//Error FB instance
EK1100_Error(
    En                  := TRUE,
    iTerminal_ID        := iTerminal_ID,
    bWcState            := FALSE,
    uiInfoData_State    := InfoData_State,
    pErrorSystem        := ErrorSystem,
    bError              => bError,
);

IF bError THEN
	sErrorMessage:=EK1100_Error.ErrorData.sErrorMessage;
ELSE
	sErrorMessage:='';
END_IF

END_FUNCTION_BLOCK

// ---- POUs/Data Type Conversion Functions/SCALE_REAL_TO_UDINT.TcPOU
FUNCTION SCALE_REAL_TO_UDINT : UDINT
VAR_INPUT
	I : REAL;
	Range_LL : REAL;
	Range_UL : REAL;
END_VAR
VAR
END_VAR

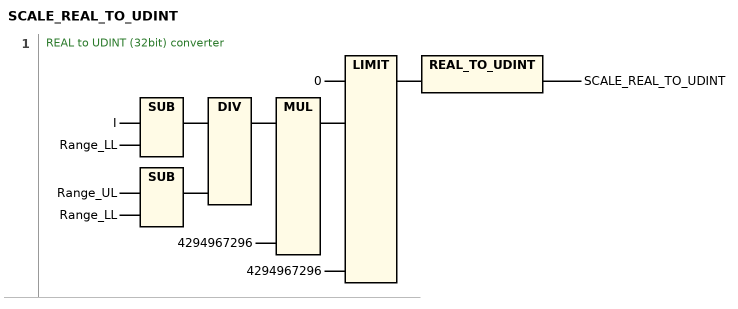
// NETWORK 1
// REAL to UDINT (32bit) converter
SCALE_REAL_TO_UDINT := REAL_TO_UDINT(LIMIT(0, ((I - Range_LL) / (Range_UL - Range_LL)) * 4294967296, 4294967296));

END_FUNCTION

// ---- POUs/Data Type Conversion Functions/SCALE_UDINT_TO_REAL.TcPOU
FUNCTION SCALE_UDINT_TO_REAL : REAL
VAR_INPUT
	I : UDINT;
	Range_LL : REAL;
	Range_UL : REAL;
END_VAR
VAR
END_VAR

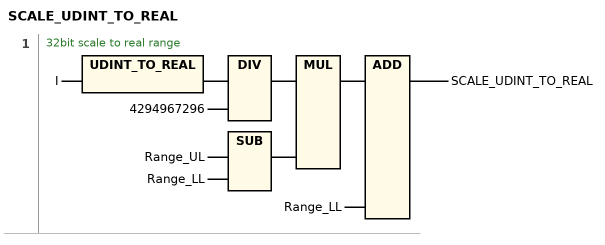
// NETWORK 1
// 32bit scale to real range
SCALE_UDINT_TO_REAL := (UDINT_TO_REAL(I) / 4294967296) * (Range_UL - Range_LL) + Range_LL;

END_FUNCTION

// ---- GlobalTextList.TcGTLO
TEXTLIST GlobalTextList
  561 = '   LocalMode'
  951 = '%2.2f'
  543 = '%2.4f'
  706 = '%i'
  940 = '%x'
  703 = 'Acknowledge'
  710 = 'Active:'
  952 = 'actPos'
  953 = 'actVel'
  110 = 'AXESMAX'
  107 = 'axisSel'
  945 = 'bBusy'
  950 = 'bBwEnabled'
  225 = 'bCommandAborted'
  946 = 'bDone'
  943 = 'bEnabled'
  941 = 'bError'
  102 = 'bExecute'
  949 = 'bFwEnabled'
  297 = 'bGeared'
  948 = 'bHomed'
  947 = 'bResetDone'
  944 = 'bWarning'
  704 = 'Clear All'
  986 = 'ehomeDirect'
  198 = 'eHomeToEncPulse_Bwd'
  510 = 'eHomeToEncPulse_Fwd'
  287 = 'eHomeToEncPulse_viaBwdLimit'
  683 = 'eHomeToEncPulse_viaFwdLimit'
  312 = 'eHomeToLimit_Bwd'
  635 = 'eHomeToLimit_Fwd'
  150 = 'eHomeToRef_Bwd'
  861 = 'eHomeToRef_Fwd'
  104 = 'ENABLE'
  106 = 'ENABLE BW'
  105 = 'ENABLE FW'
  109 = 'English'
  939 = 'errID'
  810 = 'Error #'
  705 = 'Error #:'
  702 = 'Error Log'
  707 = 'Errors:'
  768 = 'eWriteParameter'
  955 = 'fAcceleration'
  956 = 'fDeceleration'
  531 = 'fHomeFinishDistance'
  613 = 'fHomePosition'
  957 = 'fPosition'
  149 = 'fRatio'
  781 = 'fReadAxisParameter'
  708 = 'Free Entries:'
  954 = 'fVelocity'
  688 = 'fWriteAxisParameter'
  299 = 'gearIn'
  717 = 'gearInMultiMaster'
  300 = 'gearOut'
  523 = 'halt'
  566 = 'homeSensorNeg'
  677 = 'homeSensorPos'
  711 = 'Inactive:'
  116 = 'jogBw'
  117 = 'jogFw'
  298 = 'masterGear'
  111 = 'moveAbsolute'
  114 = 'moveModulo'
  113 = 'moveRelative'
  112 = 'moveVelocity'
  575 = 'nIndex'
  709 = 'Overflows:'
  942 = 'reset'
  115 = 'stop'
  108 = 'Test Language'
  103 = 'toggle'
END_TEXTLIST
